FUNCTION_BLOCK FB_PiezoDriveDS402PP EXTENDS FB_PiezoDriveDS402
VAR_INPUT
END_VAR
VAR_OUTPUT
END_VAR
VAR
    eMotionState		: 	E_DS402MotionState;
END_VAR

THIS^.Interlock();
THIS^.Power();
THIS^.DS402StateMachine();
THIS^.HandleMoveRequest();
THIS^.ReadStatus();

METHOD Brake : BOOL
SUPER^.Brake();
END_METHOD

METHOD PROTECTED ContinousMove
VAR_INPUT
END_VAR
END_METHOD

METHOD  DiscreteMove
VAR_INPUT
END_VAR
THIS^.CalibratedMotionParams();
CASE eMotionState OF
    E_DS402MotionState.PREPARE_MOTION_PARAMS:
        // Activate soft limit to avoid bumping hard on the end stops
        SUPER^.stPiezoStage.nTargetPosition := THIS^.CalibratedTargetPosition;
        SUPER^.stPiezoStage.nProfilVelocity := THIS^.CalibratedVelocity;
        SUPER^.stPiezoStage.nProfilAcceleration := THIS^.CalibratedAcceleration;
        SUPER^.stPiezoStage.nProfilDecceleration := THIS^.CalibratedAcceleration;
        SUPER^.bMoveDone := FALSE;
        SUPER^.MoveBusy := FALSE;
        SUPER^.InTargetPosition := FALSE;

        SUPER^.stPiezoStage.nModeOfOperation := E_DS402OperationMode.PROFILE_POSITION;
        eMotionState := E_DS402MotionState.INITIATE_MOTION;

    E_DS402MotionState.INITIATE_MOTION:;
        IF SUPER^.stPiezoStage.nModeOfOperationDisplay = E_DS402OperationMode.PROFILE_POSITION THEN

            // No running Job : only true for discrete motion
            IF NOT SUPER^.stPiezoStage.stPiezoDriveStatus.Bit12_OpModeSpecific THEN
                // drive dependent, it seems PI drive only support absolute motion.
                IF SUPER^.stPiezoStage.eMoveMode = E_DS402MoveMode.ABSOLUTE THEN
                    // Absolute move
                    THIS^.MoveAbsolute();
                ELSE
                    // Relative move
                    //THIS^.MoveRelative();
                END_IF
            ELSE
                //Now: we have the set point acknowledgement from the drive
                eMotionState := E_DS402MotionState.DRIVE_IN_MOTION;
            END_IF
        ELSE
            // Exit this state machine gracefully.
            eMotionState := E_DS402MotionState.DONE;
        END_IF

    E_DS402MotionState.DRIVE_IN_MOTION:;

        IF SUPER^.stPiezoStage.stPiezoDriveStatus.Bit12_OpModeSpecific THEN
            // prepare for next setpoint
            SUPER^.stPiezoStage.nPiezoDriveControl.4 := FALSE;
            SUPER^.MoveBusy := TRUE;
            eMotionState := E_DS402MotionState.TARGET_REACHED;
        END_IF

    E_DS402MotionState.TARGET_REACHED:
        IF SUPER^.stPiezoStage.stPiezoDriveStatus.TargetReached THEN
            // Halted?
            IF NOT stPiezoStage.nPiezoDriveControl.8 THEN
                THIS^.InTargetPosition := TRUE;
            ELSE
                THIS^.InTargetPosition := FALSE;
            END_IF
            // exit this state machine gracefully
            eMotionState := E_DS402MotionState.DONE;
        END_IF

    E_DS402MotionState.DONE:;
        SUPER^.bMoveDone := TRUE;
        SUPER^.MoveBusy := FALSE;
        eAxisState :=  MC_AxisStates.MC_AXISSTATE_STANDSTILL;
END_CASE

SUPER^.stPiezoStage.fPosDiff := SUPER^.stPiezoStage.fPosition - SUPER^.CalibratedActPos;
END_METHOD

METHOD DS402StateMachine
VAR_INPUT
END_VAR
SUPER^.DS402StateMachine();
END_METHOD

(*FB_Init is always available implicitly and it is used primarily for initialization.
The return value is not evaluated. For a specific influence, you can also declare the
methods explicitly and provide additional code there with the standard initialization
code. You can evaluate the return value.*)
METHOD FB_Init : BOOL
VAR_INPUT
    (* TRUE: the retain variables are initialized (reset warm / reset cold)*)
    bInitRetains	: BOOL;
    (* TRUE: the instance will be copied to the copy code afterward (online change)   *)
    bInCopyCode	: BOOL;
    stStage : REFERENCE TO ST_PiezoStage;
END_VAR
END_METHOD

METHOD Halt : BOOL
SUPER^.Halt();
END_METHOD

METHOD HandleMoveRequest : BOOL
CASE eAxisState OF

MC_AxisStates.MC_AXISSTATE_UNDEFINED:;

MC_AxisStates.MC_AXISSTATE_DISABLED:;
     // Drive back to Operation Enabled state?
    IF SUPER^.bOperational THEN
        // wait for move requests
        eAxisState :=  MC_AxisStates.MC_AXISSTATE_STANDSTILL;
    END_IF

    THIS^.bMoveBusy := FALSE;
    THIS^.bMoveDone := FALSE;
    InTargetPosition := FALSE;

MC_AxisStates.MC_AXISSTATE_STANDSTILL:
    IF SUPER^.bExecHome THEN
        eAxisState :=  MC_AxisStates.MC_AXISSTATE_HOMING;
    END_IF

    IF SUPER^.bExecMove THEN
        // we supporting only discrete motion for now
        SUPER^.stPiezoStage.nPiezoDriveControl.5 := FALSE;
        eAxisState :=  MC_AxisStates.MC_AXISSTATE_DISCRETEMOTION;
        // enter move discrete or continous here:
        eMotionState := E_DS402MotionState.PREPARE_MOTION_PARAMS;
    END_IF

    // stopping
    IF SUPER^.stPiezoStage.nPiezoDriveControl.8 THEN
        eAxisState :=  MC_AxisStates.MC_AXISSTATE_STOPPING;
    END_IF

MC_AxisStates.MC_AXISSTATE_ERRORSTOP:;
    THIS^.Reset();
    // Error Cleared?
    IF NOT SUPER^.stPiezoStage.stPiezoDriveStatus.Bit13_OpModeSpecific THEN
        eAxisState :=  MC_AxisStates.MC_AXISSTATE_UNDEFINED;
    END_IF

    THIS^.bMoveBusy := FALSE;
    THIS^.bMoveDone := FALSE;
    THIS^.InTargetPosition := FALSE;
    SUPER^.stPiezoStage.bEnable := FALSE;
    //SUPER^.bExecute := FALSE;
MC_AxisStates.MC_AXISSTATE_STOPPING:;
    eAxisState 	:= MC_AxisStates.MC_AXISSTATE_STANDSTILL;

MC_AxisStates.MC_AXISSTATE_HOMING:
    THIS^.Home();

MC_AxisStates.MC_AXISSTATE_DISCRETEMOTION:
    // bit 5: change set immediately set
    //SUPER^.stPiezoStage.nPiezoDriveControl.5 := 0;
    ContinuousMotion := FALSE;
    DiscreteMotion	:= TRUE;
    THIS^.DiscreteMove();

END_CASE

// error bit set ?
IF SUPER^.stPiezoStage.stPiezoDriveStatus.Bit13_OpModeSpecific THEN
    eAxisState :=  MC_AxisStates.MC_AXISSTATE_ERRORSTOP;
END_IF

// if the drive transition away from operational state then put the motion state mchine is disabled mode
IF NOT SUPER^.bOperational THEN
    eAxisState :=  MC_AxisStates.MC_AXISSTATE_DISABLED;
END_IF

// Check the limits and cancel execution if appropriate. Without this block we have infinite error spam
// it seems this limit are software limits.. need to be checked
IF THIS^.bMoveBusy THEN
    // Positive or Negative direction
    IF  fCalibratedStoppedPos > CalibratedActPos THEN
        THIS^.PositiveDirection := TRUE;
        THIS^.NegativeDirection := FALSE;
    ELSE
        THIS^.PositiveDirection := FALSE;
        THIS^.NegativeDirection := TRUE;
    END_IF
ELSE
    // store idle Position
    fCalibratedStoppedPos := CalibratedActPos;
END_IF

bFwdHit := THIS^.PositiveDirection AND NOT SUPER^.stPiezoStage.bAllForwardEnable;
bBwdHit := THIS^.NegativeDirection AND NOT SUPER^.stPiezoStage.bAllBackwardEnable;

IF (bFwdHit OR bBwdHit) AND NOT bHomingBusy THEN
    SUPER^.stPiezoStage.bExecute := FALSE;
END_IF

// Check done moving via user stop, fbDriveVirtual and Target Position Monitoring, or from homing.
// set/reset SUPER^.stPiezoStage.bDone after move absolute/Relative
SUPER^.ftExec(CLK:=SUPER^.stPiezoStage.bExecute);
SUPER^.rtTarget(CLK:=(THIS^.InTargetPosition AND THIS^.bMoveDone AND SUPER^.bExecMove));
SUPER^.rtHomed(CLK:=SUPER^.HomeDone AND SUPER^.bExecHome);

// user can override execute from EPICS, since we using R_TRIG on bMoveCMD this possible
IF SUPER^.ftExec.Q OR SUPER^.rtTarget.Q OR SUPER^.rtHomed.Q THEN
    IF NOT SUPER^.stPiezoStage.bDone THEN
        SUPER^.stPiezoStage.bDone := TRUE;
        SUPER^.stPiezoStage.bBusy := FALSE;
        IF NOT SUPER^.stPiezoStage.bError THEN
            SUPER^.bExecute := FALSE;
            SUPER^.stPiezoStage.bExecute := FALSE;
        END_IF
    END_IF
ELSE
    //
    SUPER^.stPiezoStage.bBusy := SUPER^.HomingBusy OR THIS^.MoveBusy;
END_IF








IF SUPER^.bExecute AND NOT stPiezoStage.bError THEN
    // Reset local warnings if things are going well
    SUPER^.stPiezoStage.sErrorMessage := '';
END_IF
END_METHOD

METHOD Home : BOOL
SUPER^.Home();
END_METHOD

METHOD Interlock : BOOL
SUPER^.Interlock();
END_METHOD

METHOD Logger : BOOL
SUPER^.Logger();
END_METHOD

METHOD MoveAbsolute

VAR

END_VAR
// Intiate the move
SUPER^.stPiezoStage.nPiezoDriveControl.6 := FALSE;
SUPER^.stPiezoStage.nPiezoDriveControl.4 := TRUE;
END_METHOD

METHOD MoveRelative
VAR_INPUT
END_VAR
// Intiate the move
SUPER^.stPiezoStage.nPiezoDriveControl.6 := TRUE;
SUPER^.stPiezoStage.nPiezoDriveControl.4 := TRUE;
END_METHOD

METHOD MoveVelocity
END_METHOD

METHOD PostMoveInterlocks
VAR_INPUT
END_VAR
// Check the limits and cancel execution if appropriate. Without this block we have infinite error spam
// it seems this limit are software limits.. need to be checked
IF THIS^.MoveBusy THEN
    // Positive or Negative direction
    IF  fCalibratedStoppedPos > CalibratedActPos THEN
        THIS^.PositiveDirection := TRUE;
        THIS^.NegativeDirection := FALSE;
    ELSE
        THIS^.PositiveDirection := FALSE;
        THIS^.NegativeDirection := TRUE;
    END_IF
ELSE
    // store idle Position
    fCalibratedStoppedPos := CalibratedActPos;
END_IF

bFwdHit := THIS^.PositiveDirection AND NOT SUPER^.stPiezoStage.bAllForwardEnable;
bBwdHit := THIS^.NegativeDirection AND NOT SUPER^.stPiezoStage.bAllBackwardEnable;

IF (bFwdHit OR bBwdHit) AND NOT bHomingBusy THEN
    SUPER^.stPiezoStage.bExecute := FALSE;
END_IF

// Check done moving via user stop, fbDriveVirtual and Target Position Monitoring, or from homing.
// set/reset SUPER^.stPiezoStage.bDone after move absolute/Relative
SUPER^.ftExec(CLK:=SUPER^.stPiezoStage.bExecute);
SUPER^.rtTarget(CLK:=(THIS^.InTargetPosition AND THIS^.MoveDone AND SUPER^.bExecMove));
SUPER^.rtHomed(CLK:=SUPER^.HomeDone AND SUPER^.bExecHome);

// user can override execute from EPICS, since we using R_TRIG on bMoveCMD this possible
IF SUPER^.ftExec.Q OR SUPER^.rtTarget.Q OR SUPER^.rtHomed.Q THEN
    IF NOT SUPER^.stPiezoStage.bDone THEN
        SUPER^.stPiezoStage.bDone := TRUE;
        SUPER^.stPiezoStage.bBusy := FALSE;
        IF NOT SUPER^.Error THEN
            SUPER^.bExecute := FALSE;
            SUPER^.stPiezoStage.bExecute := FALSE;
        END_IF
    END_IF
END_IF


IF SUPER^.bExecute AND NOT stPiezoStage.bError THEN
    // Reset local warnings if things are going well
    SUPER^.stPiezoStage.sErrorMessage := '';
END_IF
END_METHOD

METHOD Power : BOOL
SUPER^.Power();
END_METHOD

METHOD ReadStatus
SUPER^.ReadStatus();
SUPER^.SyncEpicsStatus();
END_METHOD

END_FUNCTION_BLOCK

(* stored: Version 1.1.0.1
   POU FB_PiezoDriveDS402PP: Id {6e47a4a9-16e3-49c8-8786-19fbbc700413}, SpecialFunc None
   Method Brake: Id {22a77937-1757-472e-8a24-02f41806a6fb}
   Method ContinousMove: Id {dd8dccf7-cf39-4951-959f-1329aff5f5d8}
   Method DiscreteMove: Id {0bdd1a5e-3305-4fed-8d61-3502d5d595e0}
   Method DS402StateMachine: Id {adad349e-6f22-41f6-bf4b-2c2ba773c644}
   Method FB_Init: Id {ea3b8a11-1b80-40a7-b145-7a2a5e25ca70}
   Method Halt: Id {a3eb5c8c-6142-41f2-a5f0-329f2aa7b09f}
   Method HandleMoveRequest: Id {6f021476-362f-4001-9f7a-3364b0ed4a04}
   Method Home: Id {b3172138-e5cb-4d78-92a5-25024c9364c9}
   Method Interlock: Id {ace40c54-e822-492e-bd82-afe1a2bf1748}
   Method Logger: Id {f160a88a-3c4d-4691-a405-183a03bb632e}
   Method MoveAbsolute: Id {1452777d-f00c-4295-b378-678683e81128}
   Method MoveRelative: Id {056a11cf-0783-4411-964f-fac399b96655}
   Method MoveVelocity: Id {654fd94f-9d98-4616-85f0-4b450356f9ca}
   Method PostMoveInterlocks: Id {fdfad17f-f4c5-4acf-ad7c-c467a5ef1afc}
   Method Power: Id {852126ed-4322-4881-92be-0a3202e7e349}
   Method ReadStatus: Id {f33694a7-9468-497f-90b8-80c94e8daff2} *)
